FUNCTION_BLOCK INTERNAL FINAL FB_BazMessage IMPLEMENTS I_BufferMessage

(*
syntax = "proto3";

import "tchaxx-extensions.proto";

message Foo
{
  Bar bar = 1;
  repeated Baz baz = 2 [(tchaxx.ext.v1.array_length) = 3];
}

message Bar
{
  string name = 1;
  uint32 age = 2;
  optional string email = 3;
}

message Baz
{
  fixed32 value = 1;
  string name = 2;
}
*)

VAR
	fbMessageParser : FB_MessageParser(ipMessage:= THIS^);
END_VAR

{warning 'Add method implementation '}
(* Calculates the size of this message in Protocol Buffer wire format, in bytes.*)
METHOD CalculateSize : UDINT
END_METHOD

{warning 'Add method implementation '}
METHOD InternalMergeFrom : HRESULT
VAR_IN_OUT
	stState	: ST_ParserInternalState;
END_VAR
END_METHOD

{warning 'Add method implementation '}
METHOD InternalWriteTo : HRESULT
VAR_IN_OUT
	stState	: ST_WriterInternalState;
END_VAR
END_METHOD

{warning 'Add method implementation '}
(* Merges the data from the specified coded input stream with the current message.*)
METHOD MergeFrom : HRESULT
VAR_IN_OUT
	fbInput	: FB_CodedInputStream;
END_VAR
VAR
    nTag : UDINT;
END_VAR

REPEAT   
MergeFrom := fbInput.ReadTag(nTag=>nTag);
IF SUCCEEDED(MergeFrom) AND nTag = 0 THEN
    EXIT;
END_IF;

IF FAILED(MergeFrom) THEN
    MergeFrom := MergeFrom;
    RETURN;
END_IF

CASE nTag OF
    16#0A:         // Bar bar = 1;
        fbInput.ReadRawMessage(iMessage:= THIS^);
           
 
ELSE
    MergeFrom := fBInput.SkipLastField();
END_CASE

UNTIL (FAILED(MergeFrom) OR nTag = 0)
END_REPEAT
END_METHOD

{warning 'Add property implementation'}
(* Descriptor for this message. All instances are expected to return the same descriptor,
 and for generated types this will be an explicitly-implemented member, returning the
 same value as the static property declared on the type.*)
PROPERTY MessageDescriptor : REFERENCE TO FB_MessageDescriptor
GET
END_GET
END_PROPERTY

PROPERTY PUBLIC Parser : REFERENCE TO FB_MessageParser
GET
Parser REF= THIS^.fbMessageParser;
END_GET
END_PROPERTY

{warning 'Add method implementation '}
(* Writes the data to the given coded output stream.*)
METHOD WriteTo
VAR_IN_OUT
	(* Coded output stream to write the data to. *)
	fbOutput	: FB_CodedOutputStream;
END_VAR
END_METHOD

END_FUNCTION_BLOCK

(* stored: Version 1.1.0.1
   POU FB_BazMessage: Id {98b5f4b2-3063-4e33-a1f5-a23aa9851380}, SpecialFunc None
   Method CalculateSize: Id {1c2ee7ba-a402-4ec0-b4d2-665e7c82c857}
   Method InternalMergeFrom: Id {cb841ee4-bfaf-4250-928e-6f996d90d5cb}
   Method InternalWriteTo: Id {7cc85d24-c05c-458e-9d2c-a73e9dddf506}
   Method MergeFrom: Id {01a656b6-337f-423a-a910-0aa23449dd22}
   Property MessageDescriptor: Id {0ea8b4c3-1a93-40c2-be4f-39357961749f}
   Get Get: Id {b8c4dab9-25f7-4332-b043-1d788e814c1e}
   Property Parser: Id {44ad5c3c-6e61-4f91-ad79-8466a6ade78b}
   Get Get: Id {9f4894c5-7aca-4fc0-9bb5-0e9841979a9b}
   Method WriteTo: Id {b8006ca3-cc58-474d-a5aa-598573cf89d2} *)
